{attribute addProperty BoxType "EL6201-0000-0017"}
{attribute addProperty Id "Slave_2A_DO0BIT10.1259Slave_2A_DO1BIT10.12510Slave_2A_DO2BIT10.12511Slave_2A_DO3BIT10.12512Slave_2B_DO0BIT10.12513Slave_2B_DO1BIT10.12514Slave_2B_DO2BIT10.12515Slave_2B_DO3BIT10.12516"}
{attribute addProperty CRC "3666194766"}
{attribute addProperty SizeInBites "8"}
{attribute addProperty SizeInBytes "1"}
TYPE Slave_2_Outputs_DA85B14E :
STRUCT
	{attribute addProperty Name "Slave_2A_DO0"}
	Slave_2A_DO0 : BIT;
	{attribute addProperty Name "Slave_2A_DO1"}
	Slave_2A_DO1 : BIT;
	{attribute addProperty Name "Slave_2A_DO2"}
	Slave_2A_DO2 : BIT;
	{attribute addProperty Name "Slave_2A_DO3"}
	Slave_2A_DO3 : BIT;
	{attribute addProperty Name "Slave_2B_DO0"}
	Slave_2B_DO0 : BIT;
	{attribute addProperty Name "Slave_2B_DO1"}
	Slave_2B_DO1 : BIT;
	{attribute addProperty Name "Slave_2B_DO2"}
	Slave_2B_DO2 : BIT;
	{attribute addProperty Name "Slave_2B_DO3"}
	Slave_2B_DO3 : BIT;
END_STRUCT
END_TYPE

(* stored: Version 1.2.0.0, ProductVersion 3.1.4024.9
   DUT Slave_2_Outputs_DA85B14E: Id {26e87369-774b-403b-9cbb-a047663fb69e} *)
